TYPE stComboBoxRecipes :
STRUCT
	id : INT;
	text : STRING;
	value : INT;
END_STRUCT
END_TYPE

(* stored: Version 1.1.0.1, ProductVersion 3.1.4024.13
   DUT stComboBoxRecipes: Id {fc0977b5-0e0c-4d0e-9dab-e0d6c4fb44a4} *)
